TYPE ST_CFG_DummySubsystem :
(**************************************************************************************
 * 	Application		:	BoxControl Framework
 *	Revision		:	$Revision: 404529 $
 *	Revision date	:	$Date: 2018-04-23 08:21:38 +0200 (Mo., 23 Apr 2018) $
 *	Last changed by	:	$Author: b7bolm $
 *	URL				:	$URL: http://almscdc.swisslog.com/repo/SWPD/Development/BoxControlFramework/20_Release/trunk/01_Software/BCF/BCF/JumpStart/20_Product/10_App/15_Subsystem/10_Lib/10_Conv/01_DUTs/10_Dummy/ST_CFG_DummySubsystem.TcDUT $
 *
 *	Purpose			:	Subsystem configuration
 *
 * ------------------------------------------------------------------------------------
 *	Copyright Swisslog [IP AG], Switzerland. All rights reserved.
 * 
 * ------------------------------------------------------------------------------------
 *	
 * 	Revision History: 
 *
 * 	VERSION			DATE			INITIALS			DESCRIPTION
 *	0.1				01.01.2001		swl					Example
 *
 **************************************************************************************)
STRUCT
	AM_Exists					: BOOL; // Automation manager is existing
	SPOC_Exists					: BOOL; // SPOC exists			
	tRequestReset				: TIME; // Time to reset a request
	tDelayMonitoring			: TIME; // Time to delay monitoring	
	tDelayStopping				: TIME; // Time to delay stopping
	EnableTimeSync				: BOOL; // Enable time sync
	MinTimeSync					: TIME; // Minimal time sync value
	CPU_FanExists				: BOOL; // Is true if CPU with fan equiped 
	MinFanSpeed					: UINT; // Min FAN speed
	CPU_UsageWarning			: INT; // CPU usage warning [%]
	CPU_UsageError				: INT; // CPU usage error [%]
	CPU_TemperatureWarning		: INT; // CPU temperatur warning
	CPU_TemperatureError		: INT; // CPU temperatur error
END_STRUCT
END_TYPE

(* stored: Version 1.1.0.1, ProductVersion 3.1.4022.12
   DUT ST_CFG_DummySubsystem: Id {dbe0612e-5833-4648-9f67-95291a16ccb8} *)
